FUNCTION_BLOCK FB_ControlValveStateMachine
VAR_INPUT
	controlValveCommands : ST_ExtractiveControlValveCommands;
	controlValveParameters : ST_ExtractiveControlValveParameters;
END_VAR
VAR_OUTPUT
	closeControlValve : BOOL;
	openControlValve : BOOL;
	currentControlValveOpenPercentage : DINT;
	calibrateDone : BOOL;
END_VAR
VAR
	startCalibrate : BOOL;
	RTRIG_startCalibrate : R_TRIG;
	controlState : INT;
	TOF_Calibration : TOF;
	closeCommand : BOOL;
	
	openvalve : FB_Runtime;//(resetToTime := T#0S);
	closevalve : FB_Runtime;//(resetToTime := TO_TIME(controlValveParameters.timeToFullyOpenMs));
	start : BOOL;
	setvalve : BOOL;
	open : BOOL;
	close : BOOL;
END_VAR

// Read commands from ui
startCalibrate := controlValveCommands.calibrate;
RTRIG_startCalibrate(CLK := startCalibrate);

CASE controlState OF 
	
	0: // Before calibration
		closeCommand := FALSE;
		IF RTRIG_startCalibrate.Q THEN
			controlState := 1;
		END_IF
	
	1: // Calibrate
		TOF_Calibration(IN := startCalibrate, PT := TO_TIME(controlValveParameters.calibrationTimeMs));
		startCalibrate := FALSE;
		closeCommand := TRUE;
		IF controlValveCommands.stopCalibration THEN
			TOF_Calibration(IN := FALSE);
			startCalibrate := FALSE;
			controlState := 0;
		END_IF
		IF NOT TOF_Calibration.Q THEN
			TOF_Calibration(IN := TRUE);
			calibrateDone := TRUE;
			openvalve.resetValues();
			closevalve.resetValues();
			closeCommand := FALSE;
			controlState := 2;
		END_IF
	
	2: // Control
		// Calculate how long control valve should open/close
		
		IF controlValveCommands.openPercentage > currentControlValveOpenPercentage THEN
			open := TRUE;
			close := FALSE;
		ELSIF controlValveCommands.openPercentage < currentControlValveOpenPercentage THEN
			close := FALSE;
			close := TRUE;
		ELSE
			open := FALSE;
			close := FALSE;
		END_IF
		openvalve(
				gotime := open, 
				settime := TO_TIME(controlValveParameters.timeToFullyOpenMs),
				resetToTime :=  T#0S,
				countdown := close, 
				elapsedtime => , elapsed => );
		closevalve(
				gotime := close, 
				settime := TO_TIME(controlValveParameters.timeToFullyOpenMs),
			 	resetToTime := TO_TIME(controlValveParameters.timeToFullyOpenMs),
				countdown := open, elapsedtime =>, 
				elapsed => );	
		
		// Monitor calibrate command, return to calibration step
		IF RTRIG_startCalibrate.Q THEN
			controlState := 1;
		END_IF	


END_CASE

// Calculate valve open-% according to open timer
currentControlValveOpenPercentage := TO_DINT(TIME_TO_REAL(openvalve.elapsedtime)/100);

closeControlValve := closeCommand OR close;
openControlValve := open;

END_FUNCTION_BLOCK

(* stored: Version 1.1.0.1, ProductVersion 3.1.4024.9
   POU FB_ControlValveStateMachine: Id {927e7969-28c8-49a4-a417-97545e2fb919}, SpecialFunc None *)
